% RSLogix 500 project I2P Hands-On 3 - Tanner.RSS, saved by version 10.00.00.00 %
PROJECT "UNTITLED"    % processor: Bul.1763 MicroLogix 1100 Series B %

PROGRAM FILES
  LAD 2   10 rungs

DATA FILES
  O0 OUTPUT  4 elements
  I1 INPUT  6 elements
  S2 STATUS  66 elements
  B3 BINARY  1 elements
  T4 TIMER  1 elements
  C5 COUNTER  1 elements
  R6 CONTROL  1 elements
  N7 INTEGER  1 elements
  F8 FLOAT  1 elements

LADDER 2
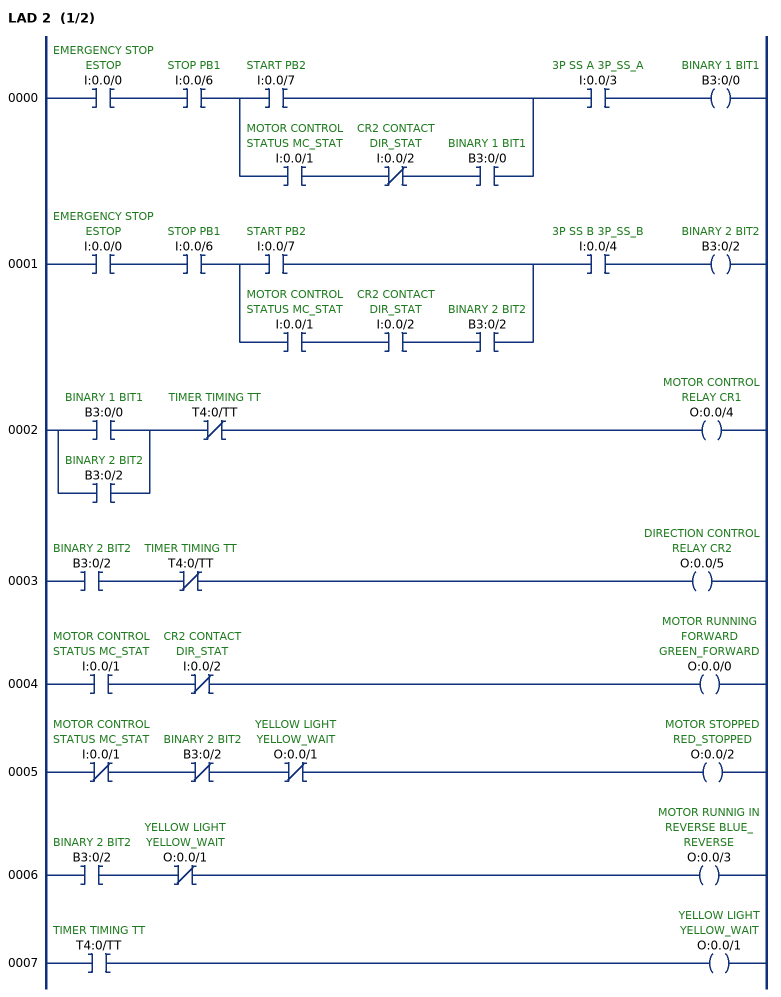
% Rung: 0 %
SOR XIC I:0.0/0 XIC I:0.0/6 BST XIC I:0.0/7 NXB XIC I:0.0/1 XIO I:0.0/2 XIC B3:0/0 BND XIC I:0.0/3 OTE B3:0/0 EOR
%   I:0.0/0  ESTOP  "EMERGENCY STOP" %
%   I:0.0/6  PB1  "STOP" %
%   I:0.0/7  PB2  "START" %
%   I:0.0/1  MC_STAT  "MOTOR CONTROL STATUS" %
%   I:0.0/2  DIR_STAT  "CR2 CONTACT" %
%   B3:0/0  BIT1  "BINARY 1" %
%   I:0.0/3  3P_SS_A  "3P SS A" %
% Rung: 1 %
SOR XIC I:0.0/0 XIC I:0.0/6 BST XIC I:0.0/7 NXB XIC I:0.0/1 XIC I:0.0/2 XIC B3:0/2 BND XIC I:0.0/4 OTE B3:0/2 EOR
%   I:0.0/0  ESTOP  "EMERGENCY STOP" %
%   I:0.0/6  PB1  "STOP" %
%   I:0.0/7  PB2  "START" %
%   I:0.0/1  MC_STAT  "MOTOR CONTROL STATUS" %
%   I:0.0/2  DIR_STAT  "CR2 CONTACT" %
%   B3:0/2  BIT2  "BINARY 2" %
%   I:0.0/4  3P_SS_B  "3P SS B" %
% Rung: 2 %
SOR BST XIC B3:0/0 NXB XIC B3:0/2 BND XIO T4:0/TT OTE O:0.0/4 EOR
%   B3:0/0  BIT1  "BINARY 1" %
%   B3:0/2  BIT2  "BINARY 2" %
%   T4:0/TT  TT  "TIMER TIMING" %
%   O:0.0/4  CR1  "MOTOR CONTROL RELAY" %
% Rung: 3 %
SOR XIC B3:0/2 XIO T4:0/TT OTE O:0.0/5 EOR
%   B3:0/2  BIT2  "BINARY 2" %
%   T4:0/TT  TT  "TIMER TIMING" %
%   O:0.0/5  CR2  "DIRECTION CONTROL RELAY" %
% Rung: 4 %
SOR XIC I:0.0/1 XIO I:0.0/2 OTE O:0.0/0 EOR
%   I:0.0/1  MC_STAT  "MOTOR CONTROL STATUS" %
%   I:0.0/2  DIR_STAT  "CR2 CONTACT" %
%   O:0.0/0  GREEN_FORWARD  "MOTOR RUNNING FORWARD" %
% Rung: 5 %
SOR XIO I:0.0/1 XIO B3:0/2 XIO O:0.0/1 OTE O:0.0/2 EOR
%   I:0.0/1  MC_STAT  "MOTOR CONTROL STATUS" %
%   B3:0/2  BIT2  "BINARY 2" %
%   O:0.0/1  YELLOW_WAIT  "YELLOW LIGHT" %
%   O:0.0/2  RED_STOPPED  "MOTOR STOPPED" %
% Rung: 6 %
SOR XIC B3:0/2 XIO O:0.0/1 OTE O:0.0/3 EOR
%   B3:0/2  BIT2  "BINARY 2" %
%   O:0.0/1  YELLOW_WAIT  "YELLOW LIGHT" %
%   O:0.0/3  BLUE_REVERSE  "MOTOR RUNNIG IN REVERSE" %
% Rung: 7 %
SOR XIC T4:0/TT OTE O:0.0/1 EOR
%   T4:0/TT  TT  "TIMER TIMING" %
%   O:0.0/1  YELLOW_WAIT  "YELLOW LIGHT" %

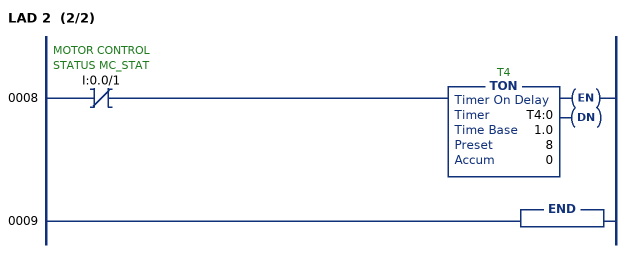
% Rung: 8 %
SOR XIO I:0.0/1 TON T4:0 1.0 8 0 EOR
%   I:0.0/1  MC_STAT  "MOTOR CONTROL STATUS" %
%   T4:0  T4 %
% Rung: 9 %
SOR END EOR

OTHER DOCUMENTED ADDRESSES
  I:0.0/5  2P_SS_POS_A  "2P SS"
  I:0.0/8  PB3  "PB3"

DATA TABLE (non-zero values as saved)
DATA T4
% .PRE .ACC %
% T4:0 % 8 0
